(* IEC 61131-3 sources: plc-home-automation/home_automation/lighting_heating_updated/src/heating, 2 files *)

(* ---- HeatingGlobals.st ---- *)
VAR_GLOBAL CONSTANT
   // Heating control locals
   C_BEDROOM_INDEX : INT            := 0;
   C_LIVING_ROOM_1_INDEX : INT      := 1;
   C_LIVING_ROOM_2_INDEX : INT      := 2;
   C_LIVING_ROOM_3_INDEX : INT      := 3;
   C_DOWNSTAIRS_BATH_INDEX : INT    := 4;
   C_HALL_INDEX : INT               := 5;
   C_GARAGE_INDEX : INT             := 6;
   C_CHILDRENS_ROOM_1_INDEX : INT   := 7;
   C_CHILDRENS_ROOM_2_INDEX : INT   := 8;
   C_CHILDRENS_ROOM_3_INDEX : INT   := 9;
   C_HALLWAY_INDEX : INT            := 10;
   C_BOILER_INDEX : INT             := 11;
   C_WC_INDEX : INT                 := 12;
   C_UPSTAIRS_BATH_INDEX : INT      := 13;
   C_HEATING_ZONES : INT            := 14;

   C_DOWNSTAIRS_ZONE_MAX_INDEX_PLUS_ONE : INT := 7;

   C_MAXIMUM_HEATING_TEMPERATURE : REAL := 38.0;
   C_MINIMUM_HEATING_TEMPERATURE : REAL := 28.0;

   C_MAXIMUM_HOT_WATER_TEMPERATURE : REAL := 62.0; // You'll need 60+ for cleaning legionella once per quarter
   C_MINIMUM_HOT_WATER_TEMPERATURE : REAL := 35.0;

END_VAR

VAR_GLOBAL
    heatingRequests : ARRAY [0 .. C_HEATING_ZONES - 1] OF BOOL;
END_VAR

VAR_GLOBAL
   HEATING_CONTROL_SAMPLING_TIME : TIME := T#10m;
   IPID_K : REAL  := 0.0005;
   IPID_TI : REAL := 0.0001;
   IPID_TD : REAL := 12000;
   OVERSHOOT_HISTERESIS : REAL := 0.2;

   HEATING_ENABLE : BOOL := true;
   HOT_WATER_ENABLE : BOOL := true;

   HOT_WATER_TEMPERATURE : REAL                 := 42.0;

   LIVING_ROOM_DESIRED_TEMPERATURE : REAL       := 22.0;
   BEDROOM_DESIRED_TEMPERATURE : REAL           := 20.5;
   CHILDRENS_ROOM_1_DESIRED_TEMPERATURE : REAL  := 22.0;
   CHILDRENS_ROOM_2_DESIRED_TEMPERATURE : REAL  := 21.0;
   CHILDRENS_ROOM_3_DESIRED_TEMPERATURE : REAL  := 21.0;
   DOWNSTAIRS_BATH_DESIRED_TEMPERATURE : REAL   := 21.0;
   UPSTAIRS_BATH_DESIRED_TEMPERATURE : REAL     := 21.0;
   GARAGE_DESIRED_TEMPERATURE : REAL            := 5.0;
   BOILER_DESIRED_TEMPERATURE : REAL            := 5.0;
   WC_DESIRED_TEMPERATURE : REAL                := 5.0;
   HALLWAY_DESIRED_TEMPERATURE : REAL           := 5.0;
   HALL_DESIRED_TEMPERATURE : REAL              := 21;

   // For testing purposes only
   // WC_TEMPERATURE : REAL              := 30.0;
   HALLWAY_TEMPERATURE : REAL         := 30.0;
   BOILER_ROOM_TEMPERATURE : REAL     := 30.0;

   SUM_HEATING_REQUIREMENT : BOOL := false;
   SUM_HEATING_WATER_TEMPERATURE_REQUIREMENT : REAL := 0;

   MEASURED_TEMPERATURES : ARRAY [0 .. C_HEATING_ZONES - 1] OF PTR_TO REAL;
   DESIRED_TEMPERATURES : ARRAY [0 .. C_HEATING_ZONES - 1] OF PTR_TO REAL;
   VALVE_ACTUATORS : ARRAY [0 .. C_HEATING_ZONES - 1] OF PTR_TO BOOL;

   // You can't take the ADR() of a real const global...
   C_50_FOK : REAL := 50.0;
   C_4_FOK : REAL  := 4.0;
END_VAR

(* ---- heating.st ---- *)
PROGRAM HeatingControl
(*Controlling Vaillant Exotec Exclusive heating bioler over VR33 OpenTherm card using tecomat OpenTherm unit.
*)

  VAR
    // Techincals for OpenThem communication
    vaillant_opentherm : fbOpenTherm;
    commEnable : BOOL := true;

    thermostats : ARRAY [0 .. C_HEATING_ZONES - 1] OF IPidHeatController;
    forwardWaterTemperatureRequests : ARRAY [0 .. C_HEATING_ZONES - 1] OF REAL;

    // Boiler heating state
    heating_start : BOOL := FALSE;

    i : INT := 0;
    activeZones : REAL := 0; // As it is an integer that will be used for division

    downstairsPumpRequest :            BOOL := FALSE;
    upstairsPumpRequest :              BOOL := FALSE;
    downstairsPumpActivationTimer :    TON;
    upstairsPumpActivationTimer :      TON;
    downstairsPumpDeactivationTimer :  TOF;
    upstairsPumpDeactivationTimer :    TOF;
    pumpActivationDelay :              TIME := T#10m;
    pumpDeactivationDelay :            TIME := T#1m;

    presenceBasedHeatingControl :      InPlaceOnOff;
    presenceBasedHotWaterControl :     InPlaceOnOff;
    heatingControlName :               STRING := 'Presence based heating control';
    hotWaterControlName :              STRING := 'Presence based hot water control';

  END_VAR

    // Actual control signals
    presenceBasedHeatingControl(requestOn := PRESENCE_BASED_HEATING_ENABLE,
                   requestOff := NOT PRESENCE_BASED_HEATING_ENABLE,
                   name := heatingControlName,
                   controlledVariable := HEATING_ENABLE);

    presenceBasedHotWaterControl(requestOn := PRESENCE_BASED_HOT_WATER_ENABLE,
                   requestOff := NOT PRESENCE_BASED_HOT_WATER_ENABLE,
                   name := hotWaterControlName,
                   controlledVariable := HOT_WATER_ENABLE);

    SUM_HEATING_REQUIREMENT := FALSE;
    downstairsPumpRequest   := FALSE;
    upstairsPumpRequest     := FALSE;
    SUM_HEATING_WATER_TEMPERATURE_REQUIREMENT := 0;
    activeZones := 0;

    // Keep heating water temperature within limits
    IF HOT_WATER_TEMPERATURE > C_MAXIMUM_HOT_WATER_TEMPERATURE THEN
       HOT_WATER_TEMPERATURE := C_MAXIMUM_HOT_WATER_TEMPERATURE;
    END_IF;

    IF HOT_WATER_TEMPERATURE < C_MINIMUM_HOT_WATER_TEMPERATURE THEN
       HOT_WATER_TEMPERATURE := C_MINIMUM_HOT_WATER_TEMPERATURE;
    END_IF;

    FOR i := 0 TO C_HEATING_ZONES - 1 DO
        // avoid unlimited accumlation of integrative error
        IF HEATING_ENABLE THEN
            thermostats[i](
                actualTemperature := MEASURED_TEMPERATURES[i]^,
                setpoint := DESIRED_TEMPERATURES[i]^,
                actualHeatingTemperature := forwardWaterTemperatureRequests[i],
                samplingTime := HEATING_CONTROL_SAMPLING_TIME,
                k := IPID_K,
                tI := IPID_TI,
                tD := IPID_TD,
                minimumHeatingTemperature := C_MINIMUM_HEATING_TEMPERATURE,
                maximumHeatingTemparature := C_MAXIMUM_HEATING_TEMPERATURE,
                overshootHisteresis := OVERSHOOT_HISTERESIS
            );
        END_IF;
        // Enable heat request for a zone only if global control flag is enabled
        heatingRequests[i] := thermostats[i].heatRequest AND HEATING_ENABLE;
        forwardWaterTemperatureRequests[i] := thermostats[i].heatingTemperature;
        SUM_HEATING_REQUIREMENT := SUM_HEATING_REQUIREMENT OR heatingRequests[i];
        IF heatingRequests[i] THEN
            SUM_HEATING_WATER_TEMPERATURE_REQUIREMENT := SUM_HEATING_WATER_TEMPERATURE_REQUIREMENT + forwardWaterTemperatureRequests[i];
            activeZones := activeZones + 1;
        END_IF;

        IF heatingRequests[i] THEN
            IF i < C_DOWNSTAIRS_ZONE_MAX_INDEX_PLUS_ONE THEN
                downstairsPumpRequest := TRUE;
            ELSE
                upstairsPumpRequest := TRUE;
            END_IF;
        END_IF;
    END_FOR;

    // Enable hall heating as an extra heatsink when downstairs bathroom heating is enabled.
    // This will help the boiler to struggle less when only 1 small room would be heated
    IF heatingRequests[C_DOWNSTAIRS_BATH_INDEX] THEN
       heatingRequests[C_HALL_INDEX] := TRUE;
    END_IF;

    IF activeZones > 0 THEN
       SUM_HEATING_WATER_TEMPERATURE_REQUIREMENT := SUM_HEATING_WATER_TEMPERATURE_REQUIREMENT / activeZones;
    END_IF;

    // Control valves
    FOR i := 0 TO C_HEATING_ZONES - 1 DO
        IF i < C_DOWNSTAIRS_ZONE_MAX_INDEX_PLUS_ONE THEN
            IF i = C_GARAGE_INDEX THEN
                // Tis is a normally closed valve
                VALVE_ACTUATORS[i]^ := heatingRequests[i] AND downstairsPumpRequest;
            ELSE
                VALVE_ACTUATORS[i]^ := NOT heatingRequests[i] AND downstairsPumpRequest;
            END_IF;
        ELSE
            VALVE_ACTUATORS[i]^ := NOT heatingRequests[i] AND upstairsPumpRequest;
        END_IF;
    END_FOR;

    downstairsPumpActivationTimer(IN := downstairsPumpRequest, PT := pumpActivationDelay);
    downstairsPumpDeactivationTimer(IN := downstairsPumpActivationTimer.Q, PT := pumpDeactivationDelay);
    upstairsPumpActivationTimer(IN := upstairsPumpRequest, PT := pumpActivationDelay);
    upstairsPumpDeactivationTimer(IN := upstairsPumpActivationTimer.Q, PT := pumpActivationDelay);

    STORAGE_PUMP := downstairsPumpDeactivationTimer.Q;
    BOILER_PUMP_PLUG_LEFT := upstairsPumpDeactivationTimer.Q;

    heating_start := downstairsPumpActivationTimer.Q OR upstairsPumpActivationTimer.Q;

    // Actual OpenTherm communication
    vaillant_opentherm(
      in_communicate := commEnable,
      in_CH_en := heating_start AND HEATING_ENABLE,
      in_DHW_en := HOT_WATER_ENABLE,
      in_CH_temp := SUM_HEATING_WATER_TEMPERATURE_REQUIREMENT,
      in_max_CH_temp := C_MAXIMUM_HEATING_TEMPERATURE,
      in_DHW_temp := HOT_WATER_TEMPERATURE,
      in_timeOut := T#10s,
      in_timeIdle := T#5s,
      UC1204_IN := void(OPENTHERM_IN),
      UC1204_OUT := void(OPENTHERM_OUT),
      OT_COMM_ARRAY := void(OT_COMM_ARRAY_GEMINOX_THRI)
    ); // Vailant Ecotec Exclusive should support all OT oiperations

    VAILLANT_ACN := vaillant_opentherm.out_ACN;
    VAILLANT_HEATING_TEMP := vaillant_opentherm.out_heating_temp;
    VAILLANT_DWH_TEMP  := vaillant_opentherm.out_DHW_temp;
    VAILLANT_OUTSIDE_TEMP := vaillant_opentherm.out_outside_temp;
    VAILLANT_RETURN_WATER_TEMP := vaillant_opentherm.out_ret_water_temp;
    VAILLANT_MODULATION_LEVEL := vaillant_opentherm.out_modulation_level;
    VAILLANT_PRESSURE_LEVEL := vaillant_opentherm.out_pressure_level;
    VAILLANT_BURNERS_RUNNING := vaillant_opentherm.out_burner_starts;
    VAILLANT_HEATING_ACTIVE := vaillant_opentherm.out_CH_active;
    VAILLANT_DWH_ACTIVE := vaillant_opentherm.out_DHW_active;
    VAILANT_DWH_PRESENT := vaillant_opentherm.out_DHW_present;
    VAILANT_MODULATION_SUPPORT := vaillant_opentherm.out_modulating;
    VAILANT_BURNER_ON := vaillant_opentherm.out_flame;
    VAILANT_ERROR := vaillant_opentherm.out_com_error;
    VAILLANT_DIAG_CODE := vaillant_opentherm.out_diag_code;
    VAILANT_COMMUNICATIONO_ERROR := vaillant_opentherm.out_com_error;

END_PROGRAM
